Staubli VAL3: tRobot.pgx

program tRobot()
  local num l_nIdx
begin
  resetMotion(jStart)

  while !bFinish
    // Attente qu il y ait au moins un point dans la file
    wait(nQueueCount > 0)

    // Lecture du point courant dans la file
    l_nIdx = nQueueRead

    // Verification continuite des trames
    if nIndexQueue[l_nIdx] == nLastIndex + 1

      // Configuration vitesse pour ce point
      mNomSpeed.vel = nVelQueue[l_nIdx]
      pCmdQueue[l_nIdx].config.shoulder = lefty
      pCmdQueue[l_nIdx].config.wrist    = wpositive
      pCmdQueue[l_nIdx].config.elbow    = epositive
      logMsg("Point: x=" + toString(".1", pCmdQueue[l_nIdx].trsf.x) + " y=" + toString(".1", pCmdQueue[l_nIdx].trsf.y) + " z=" + toString(".1", pCmdQueue[l_nIdx].trsf.z))

      // Execution du mouvement selon le type
      if nTypeQueue[l_nIdx] == 0
        movel(pCmdQueue[l_nIdx], tBuse, mNomSpeed)
      else
        movel(pCmdQueue[l_nIdx], tBuse, mNomSpeed)
      endIf
      waitEndMove()

      nLastIndex = nIndexQueue[l_nIdx]

      // Envoi ACK + etat file : {ACK;index_execute;n_restant}
      sAck = "{ACK;" + toString("", nLastIndex) + ";" + toString("", nQueueCount) + "}"
      nAckIndex = 0
      while nAckIndex < len(sAck)
        sioSet(sioSocket, asc(sAck, nAckIndex))
        nAckIndex = nAckIndex + 1
      endWhile
      sioSet(sioSocket, nEol)

    else
      logMsg("Erreur trame, attendue: " + toString("", nLastIndex+1) + " recue: " + toString("", nIndexQueue[l_nIdx]))
      nLastIndex = nIndexQueue[l_nIdx] - 1
    endIf

    // Avance le pointeur de lecture
    nQueueRead = nQueueRead + 1
    if nQueueRead >= nQueueSize
      nQueueRead = 0
    endIf
    nQueueCount = nQueueCount - 1

    delay(0)
  endWhile

  waitEndMove()
end
